PROGRAM P02_P2P
VAR
END_VAR

//P2P_ST300_MODBUS();
P2P_LH();
P2P_TB();

END_PROGRAM

(* stored: Version 1.1.0.1, ProductVersion 3.1.4024.12
   POU P02_P2P: Id {65144f6b-0d8b-41ed-8fc7-ccd91a54ba08}, SpecialFunc None *)
